FUNCTION_BLOCK FB_SealStages

VAR_INPUT
	Axis 			: AXIS_REF; //Reference for the axis configured in the AX8108
    iTargetPosition : INT; 		//Target motor position
    rVelocity 		: LREAL; 	//Motor velocity
    rAcceleration 	: LREAL; 	//Motor acceleration
    rDeceleration 	: LREAL; 	//Motor deceleration
    bExecute 		: BOOL;  	//Start the movement
END_VAR

VAR_OUTPUT
	bSealSucess 	: BOOL; 	//Indicates whether the process was completed successfully
    bSealError 		: BOOL;  	//Indicates whether there was an error during execution
END_VAR

VAR
	MotorStageCollection 	: FB_StageCollectionMotor; 	
	MotorAxis 				: AXIS_REF;                 //FB instance for the motor
    MotorInPosition 		: BOOL;                     //Flag to indicate position reached
    MotorBusy 				: BOOL;                     //Flag to indicate movement in progress
    MotorError 				: BOOL;                     //Flag to indicate error
    MotorErrorID 			: UDINT; 
	
	FB_GetPosition		: FB_GetPosition;
		bGetPosition	: BOOL := FALSE;
	
	FB_MotorControl		: FB_MotorControl;
		bMoveDone		: BOOL := FALSE;
		bPosError		: BOOL := FALSE;
		nPosErrorID		: UDINT;
		sState			: STRING(256);
				
	fbSetZero			: MC_SetPosition;
	
	fbReadStatus		: MC_ReadStatus;
END_VAR

//Geting the M1 Motor actual position
IF bGetPosition THEN	
	FB_GetPosition(
		bEnable		:=	TRUE,
		AxisRef		:=	Axis,
		bError		=>	bPosError,
		nErrorID	=>	nPosErrorID,
		rPosition	=>	GVL_Motion.M1Motor.rActualPosition
	);		
END_IF

IF GVL_Motion.M1Motor.rActualPosition <> iTargetPosition THEN
	//Motor M1 Moving FB
	IF bExecute AND GVL_Safety.iMotorsSTOEnabled THEN
		FB_MotorControl(
			bEnable 	:= TRUE,
			AxisRef 	:= Axis, 
			nPosition 	:= iTargetPosition, 
			nVelocity 	:= rVelocity,
			bDone		=> bMoveDone,
			bError		=> bPosError,
			nErrorID	=> nPosErrorID,
			sState		=> sState
		);
	END_IF
		
	IF MotorStageCollection.Error THEN
		//Indicate Error
		bSealError 	:= TRUE;
		bSealSucess := FALSE;
	ELSE
		bSealError 	:= FALSE;
		IF MotorStageCollection.InPosition THEN
			//Sucess return boolean
			bSealSucess := TRUE;
		ELSE
			bSealSucess := FALSE;
		END_IF;
	END_IF;
END_IF

END_FUNCTION_BLOCK

(* stored: Version 1.1.0.1, ProductVersion 3.1.4024.12
   POU FB_SealStages: Id {b9c49897-ef39-427d-b9c0-f5c61609c2a7}, SpecialFunc None *)
